// TIA Portal V19 program export: 1 tag tables, 0 data types, 3 data blocks, 3 code blocks (in call order from the OBs), 0 instance data blocks

VAR_GLOBAL   // PLC tag table "Default tag table"
   RHSystemClockByte AT %IB0 : Byte;   // Recieved from RH System as heartbeat
   InputByte1 AT %IB1 : Byte;
   InputByte2 AT %IB2 : Byte;
   InputByte3 AT %IB3 : Byte;
   InputByte4 AT %IB4 : Byte;
   InputByte5 AT %IB5 : Byte;
   InputByte6 AT %IB6 : Byte;
   InputByte7 AT %IB7 : Byte;
   InputByte8 AT %IB8 : Byte;
   InputByte9 AT %IB9 : Byte;
   InputByte10 AT %IB10 : Byte;
   LocalSystemClockbyte AT %QB0 : Byte;   // Sent to RH System as heartbeat
   OutputByte1 AT %QB1 : Byte;
   OutputByte2 AT %QB2 : Byte;
   OutputByte3 AT %QB3 : Byte;
   OutputByte4 AT %QB4 : Byte;
   OutputByte5 AT %QB5 : Byte;
   OutputByte6 AT %QB6 : Byte;
   OutputByte7 AT %QB7 : Byte;
   OutputByte8 AT %QB8 : Byte;
   OutputByte9 AT %QB9 : Byte;
   OutputByte10 AT %QB10 : Byte;
   System_Byte AT %MB1 : Byte;
   FirstScan AT %M1.0 : Bool;
   DiagStatusUpdate AT %M1.1 : Bool;
   AlwaysTRUE AT %M1.2 : Bool;
   AlwaysFALSE AT %M1.3 : Bool;
   Clock_Byte AT %MB0 : Byte;
   Clock_10Hz AT %M0.0 : Bool;
   Clock_5Hz AT %M0.1 : Bool;
   "Clock_2.5Hz" AT %M0.2 : Bool;
   Clock_2Hz AT %M0.3 : Bool;
   "Clock_1.25Hz" AT %M0.4 : Bool;
   Clock_1Hz AT %M0.5 : Bool;
   "Clock_0.625Hz" AT %M0.6 : Bool;
   "Clock_0.5Hz" AT %M0.7 : Bool;
   GreenPushButton AT %IB27 : Byte;
   BluePushButton AT %IB34 : Byte;
   SelectorSwitch AT %IB35 : Byte;
   RedPushButton AT %IB36 : Byte;
   GreenPushButtonLamp AT %QB32 : Byte;
   BluePushButtonLamp AT %QB33 : Byte;
   SelectorSwitchLamp AT %QB34 : Byte;
   RedPushButtonLamp AT %QB35 : Byte;
   "EstopF-In_ModuleByte1" AT %IB28 : Byte;
   "EstopF-In_ModuleByte2" AT %IB29 : Byte;
   "EstopF-In_ModuleByte3" AT %IB30 : Byte;
   "EstopF-In_ModuleByte4" AT %IB31 : Byte;
   "EstopF-In_ModuleByte5" AT %IB32 : Byte;
   "EstopF-In_ModuleByte6" AT %IB33 : Byte;
   "Estop-FOut_ModuleByte1" AT %QB28 : Byte;
   "Estop-FOut_ModuleByte2" AT %QB29 : Byte;
   "Estop-FOut_ModuleByte3" AT %QB30 : Byte;
   "Estop-FOut_ModuleByte4" AT %QB31 : Byte;
END_VAR

DATA_BLOCK "PLCGlobal_DB"   // DB3
{ S7_Optimized_Access := 'TRUE' }
// stored: MemoryReserve 100
   VAR
      SafetyAckReset : Bool;
      GreenLampProcessActive : Bool;
      BluePushButton : Bool;
      SelectorSwitch : Bool;
      RedPushButton : Bool;
      GreenPushButtonLamp : Bool;
      BluePushButtonLamp : Bool;
      SelectorSwitchLamp : Bool;
      RedPushButtonLamp : Bool;
   END_VAR
BEGIN
END_DATA_BLOCK

DATA_BLOCK "GlobalSafetyDB"   // DB6, F_DB
{ S7_Optimized_Access := 'TRUE' }
   VAR
      GlobalEstop : Bool;
      GlobalAck : Bool;   // Used to acknowledge global failsafety
      SubordinateEstop : Bool;
      ClockByteSupervisory : Int;
   END_VAR
BEGIN
END_DATA_BLOCK

DATA_BLOCK "SafetyDataExchangeDB"   // DB7
{ S7_Optimized_Access := 'TRUE' }
// stored: MemoryReserve 100
   VAR
      SubordinateClockByte : Int;
   END_VAR
BEGIN
END_DATA_BLOCK

ORGANIZATION_BLOCK "Main"   // OB1, LAD, ProgramCycle
TITLE = "Main Program Sweep (Cycle)"
{ S7_Optimized_Access := 'TRUE' }
// stored: SetENOAutomatically false
   VAR_INPUT
      Initial_Call : Bool;   // Initial call of this OB
      Remanence : Bool;   // =True, if remanent data are available
   END_VAR
BEGIN

REGION Network 1: Write clockbyte out to RH System, Display RH System clock byte inline
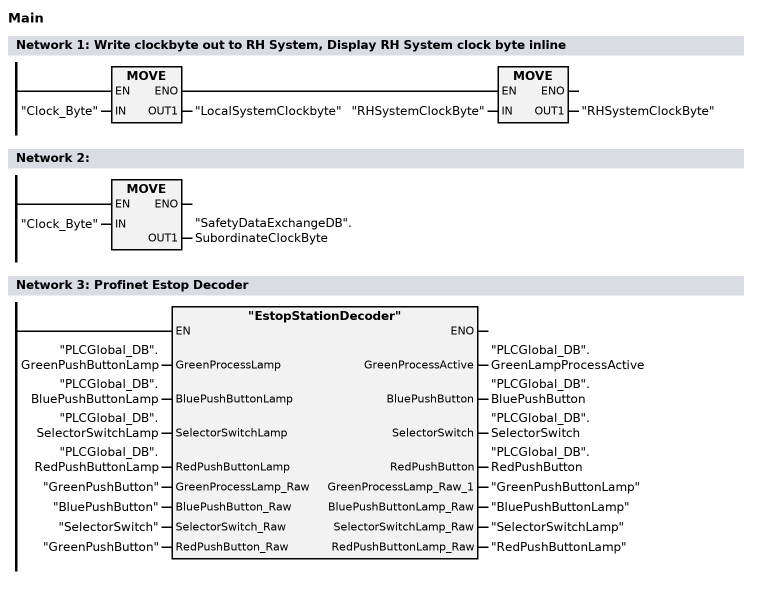
   RUNG wire#powerrail
      Move(in := "Clock_Byte", out1 => "LocalSystemClockbyte")
      Move(in := "RHSystemClockByte", out1 => "RHSystemClockByte")
   END_RUNG
   // the same network as SCL:
   "LocalSystemClockbyte" := "Clock_Byte";
   "RHSystemClockByte" := "RHSystemClockByte";
END_REGION

REGION Network 2
   RUNG wire#powerrail
      Move(in := "Clock_Byte", out1 => "SafetyDataExchangeDB".SubordinateClockByte)
   END_RUNG
   // the same network as SCL:
   "SafetyDataExchangeDB".SubordinateClockByte := "Clock_Byte";
END_REGION

REGION Network 3: Profinet Estop Decoder
   RUNG wire#powerrail
      "EstopStationDecoder"(GreenProcessLamp := "PLCGlobal_DB".GreenPushButtonLamp, BluePushButtonLamp := "PLCGlobal_DB".BluePushButtonLamp, SelectorSwitchLamp := "PLCGlobal_DB".SelectorSwitchLamp, RedPushButtonLamp := "PLCGlobal_DB".RedPushButtonLamp, GreenProcessLamp_Raw := "GreenPushButton", BluePushButton_Raw := "BluePushButton", SelectorSwitch_Raw := "SelectorSwitch", RedPushButton_Raw := "GreenPushButton", GreenProcessActive => "PLCGlobal_DB".GreenLampProcessActive, BluePushButton => "PLCGlobal_DB".BluePushButton, SelectorSwitch => "PLCGlobal_DB".SelectorSwitch, RedPushButton => "PLCGlobal_DB".RedPushButton, GreenProcessLamp_Raw_1 => "GreenPushButtonLamp", BluePushButtonLamp_Raw => "BluePushButtonLamp", SelectorSwitchLamp_Raw => "SelectorSwitchLamp", RedPushButtonLamp_Raw => "RedPushButtonLamp")
   END_RUNG
   // the same network as SCL:
   "EstopStationDecoder"(GreenProcessLamp := "PLCGlobal_DB".GreenPushButtonLamp,
                         BluePushButtonLamp := "PLCGlobal_DB".BluePushButtonLamp,
                         SelectorSwitchLamp := "PLCGlobal_DB".SelectorSwitchLamp,
                         RedPushButtonLamp := "PLCGlobal_DB".RedPushButtonLamp,
                         GreenProcessLamp_Raw := "GreenPushButton",
                         BluePushButton_Raw := "BluePushButton",
                         SelectorSwitch_Raw := "SelectorSwitch",
                         RedPushButton_Raw := "GreenPushButton",
                         GreenProcessActive => "PLCGlobal_DB".GreenLampProcessActive,
                         BluePushButton => "PLCGlobal_DB".BluePushButton,
                         SelectorSwitch => "PLCGlobal_DB".SelectorSwitch,
                         RedPushButton => "PLCGlobal_DB".RedPushButton,
                         GreenProcessLamp_Raw_1 => "GreenPushButtonLamp",
                         BluePushButtonLamp_Raw => "BluePushButtonLamp",
                         SelectorSwitchLamp_Raw => "SelectorSwitchLamp",
                         RedPushButtonLamp_Raw => "RedPushButtonLamp");
END_REGION
END_ORGANIZATION_BLOCK

FUNCTION "EstopStationDecoder" : Void   // FC1, LAD
{ S7_Optimized_Access := 'TRUE' }
// stored: SetENOAutomatically false
   VAR_INPUT
      GreenProcessLamp : Bool;
      BluePushButtonLamp : Bool;
      SelectorSwitchLamp : Bool;
      RedPushButtonLamp : Bool;
      GreenProcessLamp_Raw : Byte;
      BluePushButton_Raw : Byte;
      SelectorSwitch_Raw : Byte;
      RedPushButton_Raw : Byte;
   END_VAR
   VAR_OUTPUT
      GreenProcessActive : Bool;
      BluePushButton : Bool;
      SelectorSwitch : Bool;
      RedPushButton : Bool;
      GreenProcessLamp_Raw_1 : Byte;
      BluePushButtonLamp_Raw : Byte;
      SelectorSwitchLamp_Raw : Byte;
      RedPushButtonLamp_Raw : Byte;
   END_VAR
BEGIN

REGION Network 1: Profinet Estop Decoder
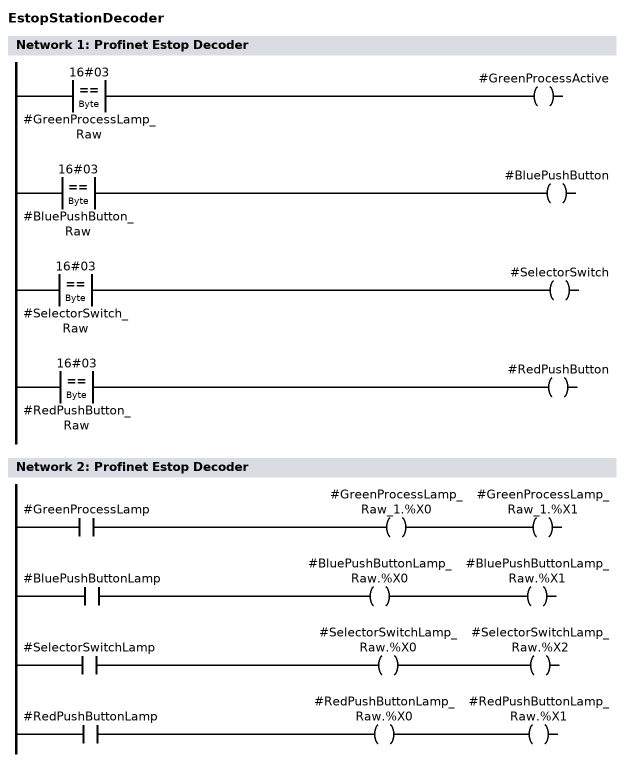
   RUNG wire#powerrail
      { S7_Templates := "SrcType := Byte" } EQ_Contact(in1 := 16#03, in2 := #GreenProcessLamp_Raw)
      Coil( #GreenProcessActive )
   END_RUNG
   RUNG wire#powerrail
      { S7_Templates := "SrcType := Byte" } EQ_Contact(in1 := 16#03, in2 := #BluePushButton_Raw)
      Coil( #BluePushButton )
   END_RUNG
   RUNG wire#powerrail
      { S7_Templates := "SrcType := Byte" } EQ_Contact(in1 := 16#03, in2 := #SelectorSwitch_Raw)
      Coil( #SelectorSwitch )
   END_RUNG
   RUNG wire#powerrail
      { S7_Templates := "SrcType := Byte" } EQ_Contact(in1 := 16#03, in2 := #RedPushButton_Raw)
      Coil( #RedPushButton )
   END_RUNG
   // the same network as SCL:
   #GreenProcessActive := 16#03 = #GreenProcessLamp_Raw;
   #BluePushButton := 16#03 = #BluePushButton_Raw;
   #SelectorSwitch := 16#03 = #SelectorSwitch_Raw;
   #RedPushButton := 16#03 = #RedPushButton_Raw;
END_REGION

REGION Network 2: Profinet Estop Decoder
   RUNG wire#powerrail
      Contact( #GreenProcessLamp )
      Coil( #GreenProcessLamp_Raw_1.%X0 )
      Coil( #GreenProcessLamp_Raw_1.%X1 )
   END_RUNG
   RUNG wire#powerrail
      Contact( #BluePushButtonLamp )
      Coil( #BluePushButtonLamp_Raw.%X0 )
      Coil( #BluePushButtonLamp_Raw.%X1 )
   END_RUNG
   RUNG wire#powerrail
      Contact( #SelectorSwitchLamp )
      Coil( #SelectorSwitchLamp_Raw.%X0 )
      Coil( #SelectorSwitchLamp_Raw.%X2 )
   END_RUNG
   RUNG wire#powerrail
      Contact( #RedPushButtonLamp )
      Coil( #RedPushButtonLamp_Raw.%X0 )
      Coil( #RedPushButtonLamp_Raw.%X1 )
   END_RUNG
   // the same network as SCL:
   #GreenProcessLamp_Raw_1.%X0 := #GreenProcessLamp;
   #GreenProcessLamp_Raw_1.%X1 := #GreenProcessLamp;
   #BluePushButtonLamp_Raw.%X0 := #BluePushButtonLamp;
   #BluePushButtonLamp_Raw.%X1 := #BluePushButtonLamp;
   #SelectorSwitchLamp_Raw.%X0 := #SelectorSwitchLamp;
   #SelectorSwitchLamp_Raw.%X2 := #SelectorSwitchLamp;
   #RedPushButtonLamp_Raw.%X0 := #RedPushButtonLamp;
   #RedPushButtonLamp_Raw.%X1 := #RedPushButtonLamp;
END_REGION
END_FUNCTION

FUNCTION_BLOCK "Main_Safety_RTG1"   // FB1, F_LAD
{ S7_Optimized_Access := 'TRUE' }
// stored: AutoNumber false
   VAR_TEMP
      EstopLamp : Bool;
   END_VAR
   VAR_TEMP   // added for the SCL form of the ladder/FBD networks
      _w1 : Bool;
   END_VAR
BEGIN

REGION Network 1
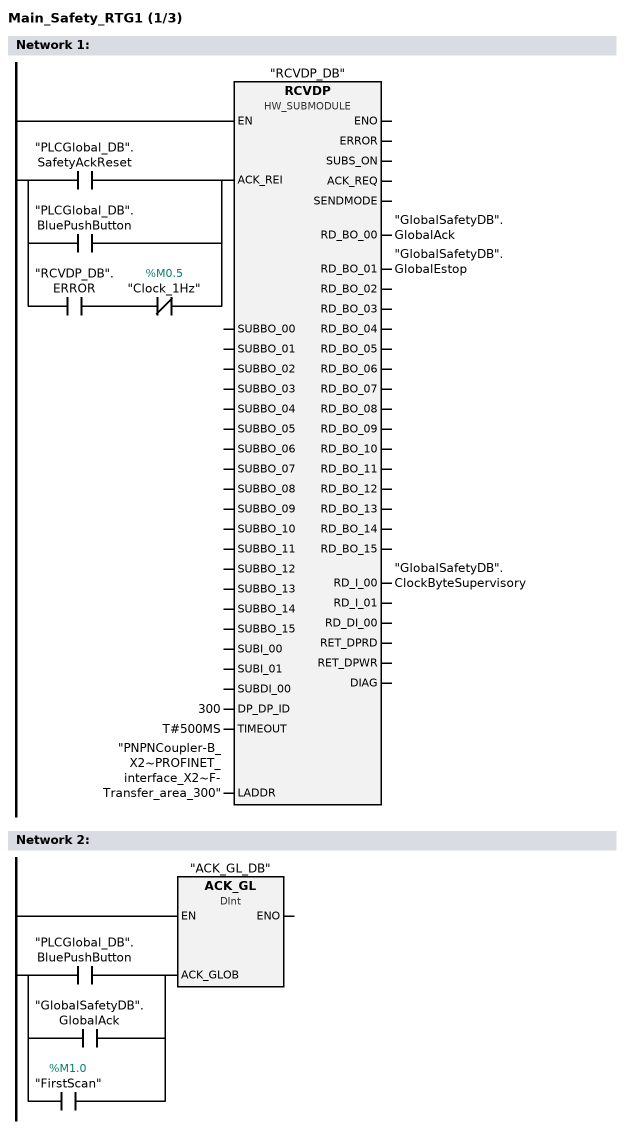
   RUNG wire#powerrail
      { S7_Templates := "laddr_type := HW_SUBMODULE" } "RCVDP_DB".RCVDP(ACK_REI := wire#w1, SUBBO_00 :=, SUBBO_01 :=, SUBBO_02 :=, SUBBO_03 :=, SUBBO_04 :=, SUBBO_05 :=, SUBBO_06 :=, SUBBO_07 :=, SUBBO_08 :=, SUBBO_09 :=, SUBBO_10 :=, SUBBO_11 :=, SUBBO_12 :=, SUBBO_13 :=, SUBBO_14 :=, SUBBO_15 :=, SUBI_00 :=, SUBI_01 :=, SUBDI_00 :=, DP_DP_ID := 300, TIMEOUT := T#500MS, LADDR := "PNPNCoupler-B_X2~PROFINET_interface_X2~F-Transfer_area_300", ERROR =>, SUBS_ON =>, ACK_REQ =>, SENDMODE =>, RD_BO_00 => "GlobalSafetyDB".GlobalAck, RD_BO_01 => "GlobalSafetyDB".GlobalEstop, RD_BO_02 =>, RD_BO_03 =>, RD_BO_04 =>, RD_BO_05 =>, RD_BO_06 =>, RD_BO_07 =>, RD_BO_08 =>, RD_BO_09 =>, RD_BO_10 =>, RD_BO_11 =>, RD_BO_12 =>, RD_BO_13 =>, RD_BO_14 =>, RD_BO_15 =>, RD_I_00 => "GlobalSafetyDB".ClockByteSupervisory, RD_I_01 =>, RD_DI_00 =>, RET_DPRD =>, RET_DPWR =>, DIAG =>)
   END_RUNG
   RUNG wire#powerrail
      Contact( "PLCGlobal_DB".SafetyAckReset )
   END_RUNG wire#w1
   RUNG wire#powerrail
      Contact( "PLCGlobal_DB".BluePushButton )
   END_RUNG wire#w1
   RUNG wire#powerrail
      Contact( "RCVDP_DB".ERROR )
      I_Contact( "Clock_1Hz" )
   END_RUNG wire#w1
   // the same network as SCL:
   "RCVDP_DB"(ACK_REI := "PLCGlobal_DB".SafetyAckReset OR "PLCGlobal_DB".BluePushButton OR ("RCVDP_DB".ERROR AND NOT "Clock_1Hz"),   // RCVDP
              DP_DP_ID := 300,
              TIMEOUT := T#500MS,
              LADDR := "PNPNCoupler-B_X2~PROFINET_interface_X2~F-Transfer_area_300",
              RD_BO_00 => "GlobalSafetyDB".GlobalAck,
              RD_BO_01 => "GlobalSafetyDB".GlobalEstop,
              RD_I_00 => "GlobalSafetyDB".ClockByteSupervisory);
END_REGION

REGION Network 2
   RUNG wire#powerrail
      { S7_Templates := "codedbool_type := DInt" } "ACK_GL_DB".ACK_GL(ACK_GLOB := wire#w1)
   END_RUNG
   RUNG wire#powerrail
      Contact( "PLCGlobal_DB".BluePushButton )
   END_RUNG wire#w1
   RUNG wire#powerrail
      Contact( "GlobalSafetyDB".GlobalAck )
   END_RUNG wire#w1
   RUNG wire#powerrail
      Contact( "FirstScan" )
   END_RUNG wire#w1
   // the same network as SCL:
   "ACK_GL_DB"(ACK_GLOB := "PLCGlobal_DB".BluePushButton OR "GlobalSafetyDB".GlobalAck OR "FirstScan");   // ACK_GL
END_REGION

REGION Network 3
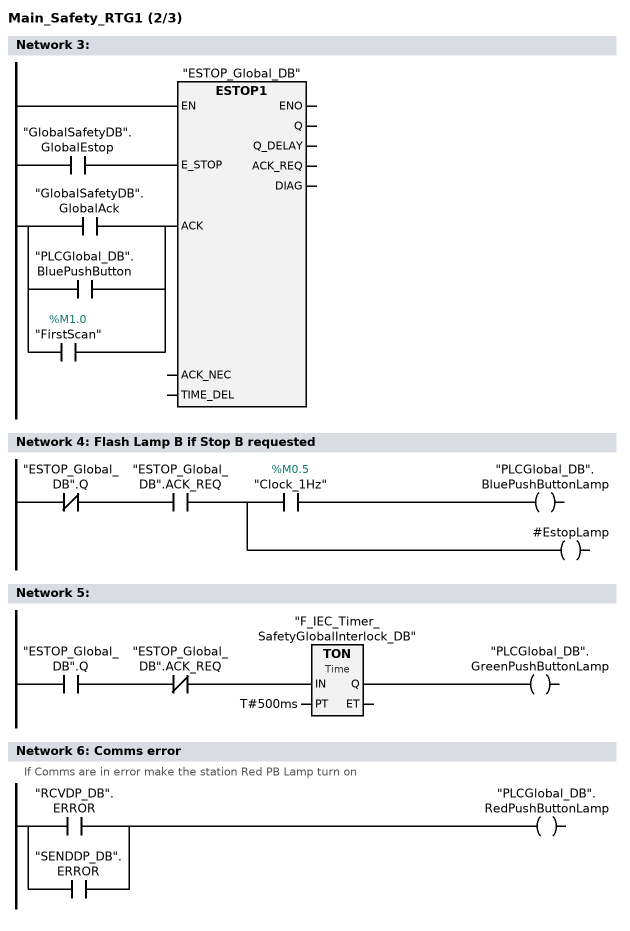
   RUNG wire#powerrail
      "ESTOP_Global_DB".ESTOP1(E_STOP := wire#w1, ACK := wire#w2, ACK_NEC :=, TIME_DEL :=, Q =>, Q_DELAY =>, ACK_REQ =>, DIAG =>)
   END_RUNG
   RUNG wire#powerrail
      Contact( "GlobalSafetyDB".GlobalEstop )
   END_RUNG wire#w1
   RUNG wire#powerrail
      Contact( "GlobalSafetyDB".GlobalAck )
   END_RUNG wire#w2
   RUNG wire#powerrail
      Contact( "PLCGlobal_DB".BluePushButton )
   END_RUNG wire#w2
   RUNG wire#powerrail
      Contact( "FirstScan" )
   END_RUNG wire#w2
   // the same network as SCL:
   "ESTOP_Global_DB"(E_STOP := "GlobalSafetyDB".GlobalEstop,   // ESTOP1
                     ACK := "GlobalSafetyDB".GlobalAck OR "PLCGlobal_DB".BluePushButton OR "FirstScan");
END_REGION

REGION Network 4: Flash Lamp B if Stop B requested
   RUNG wire#powerrail
      I_Contact( "ESTOP_Global_DB".Q )
      Contact( "ESTOP_Global_DB".ACK_REQ )
      wire#w1
      Contact( "Clock_1Hz" )
      Coil( "PLCGlobal_DB".BluePushButtonLamp )
   END_RUNG
   RUNG wire#w1
      Coil( #EstopLamp )
   END_RUNG
   // the same network as SCL:
   #_w1 := NOT "ESTOP_Global_DB".Q AND "ESTOP_Global_DB".ACK_REQ;
   "PLCGlobal_DB".BluePushButtonLamp := #_w1 AND "Clock_1Hz";
   #EstopLamp := #_w1;
END_REGION

REGION Network 5
   RUNG wire#powerrail
      Contact( "ESTOP_Global_DB".Q )
      I_Contact( "ESTOP_Global_DB".ACK_REQ )
      { S7_Templates := "[time_type := Time, codedbool_type := DInt]" } "F_IEC_Timer_SafetyGlobalInterlock_DB".TON(pt := T#500ms, et =>)
      Coil( "PLCGlobal_DB".GreenPushButtonLamp )
   END_RUNG
   // the same network as SCL:
   "F_IEC_Timer_SafetyGlobalInterlock_DB".TON(IN := "ESTOP_Global_DB".Q AND NOT "ESTOP_Global_DB".ACK_REQ,
                           PT := T#500ms);
   "PLCGlobal_DB".GreenPushButtonLamp := "F_IEC_Timer_SafetyGlobalInterlock_DB".Q;
END_REGION

REGION Network 6: Comms error
   // If Comms are in error make the station Red PB Lamp turn on
   RUNG wire#powerrail
      Contact( "RCVDP_DB".ERROR )
      wire#w1
      Coil( "PLCGlobal_DB".RedPushButtonLamp )
   END_RUNG
   RUNG wire#powerrail
      Contact( "SENDDP_DB".ERROR )
   END_RUNG wire#w1
   // the same network as SCL:
   "PLCGlobal_DB".RedPushButtonLamp := "RCVDP_DB".ERROR OR "SENDDP_DB".ERROR;
END_REGION

REGION Network 7
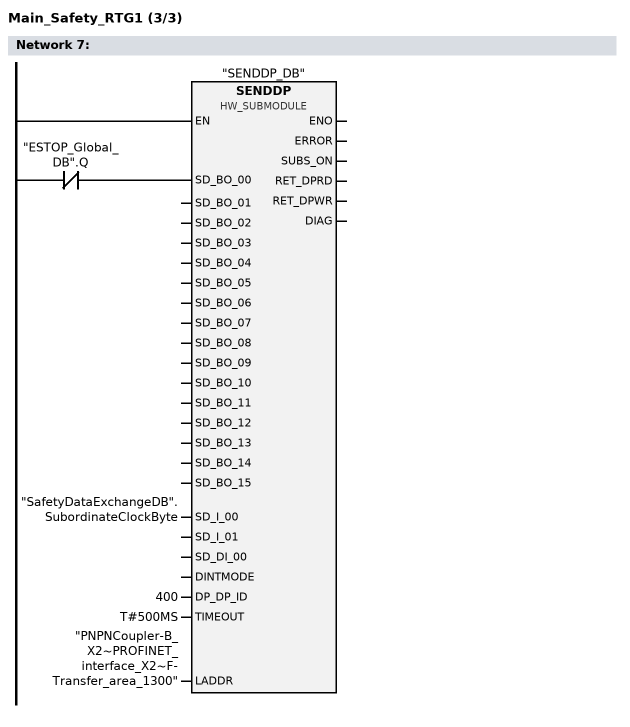
   RUNG wire#powerrail
      { S7_Templates := "laddr_type := HW_SUBMODULE" } "SENDDP_DB".SENDDP(SD_BO_00 := wire#w1, SD_BO_01 :=, SD_BO_02 :=, SD_BO_03 :=, SD_BO_04 :=, SD_BO_05 :=, SD_BO_06 :=, SD_BO_07 :=, SD_BO_08 :=, SD_BO_09 :=, SD_BO_10 :=, SD_BO_11 :=, SD_BO_12 :=, SD_BO_13 :=, SD_BO_14 :=, SD_BO_15 :=, SD_I_00 := "SafetyDataExchangeDB".SubordinateClockByte, SD_I_01 :=, SD_DI_00 :=, DINTMODE :=, DP_DP_ID := 400, TIMEOUT := T#500MS, LADDR := "PNPNCoupler-B_X2~PROFINET_interface_X2~F-Transfer_area_1300", ERROR =>, SUBS_ON =>, RET_DPRD =>, RET_DPWR =>, DIAG =>)
   END_RUNG
   RUNG wire#powerrail
      I_Contact( "ESTOP_Global_DB".Q )
   END_RUNG wire#w1
   // the same network as SCL:
   "SENDDP_DB"(SD_BO_00 := NOT "ESTOP_Global_DB".Q,   // SENDDP
               SD_I_00 := "SafetyDataExchangeDB".SubordinateClockByte,
               DP_DP_ID := 400,
               TIMEOUT := T#500MS,
               LADDR := "PNPNCoupler-B_X2~PROFINET_interface_X2~F-Transfer_area_1300");
END_REGION
END_FUNCTION_BLOCK
